PROGRAM Auswertung
VAR
END_VAR

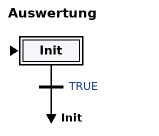
INITIAL_STEP Init:
END_STEP
TRANSITION FROM Init TO Init
    := TRUE;
END_TRANSITION

END_PROGRAM

(* stored: Version 1.1.0.1, ProductVersion 3.1.4024.12
   POU Auswertung: Id {ad7635de-101d-4726-9f88-612ab6d15e20}, SpecialFunc None *)
